TYPE ST_ParFilterAD :  //P1部分参数
STRUCT
	iLimitH             :REAL;//转换前高限值
	iLimitL             :REAL;//转换前低限值
	fRangeH         :REAL;//量程高限
	fRangeL          :REAL;//量程低限
END_STRUCT
END_TYPE

(* stored: Version 1.1.0.1, ProductVersion 3.1.4024.9
   DUT ST_ParFilterAD: Id {3a45f496-ee49-4698-8c76-b929c7d4132c} *)
